FUNCTION_BLOCK TcContinuousAxisCommand IMPLEMENTS itfContinuousAxisCommand
VAR_INPUT
END_VAR
VAR_OUTPUT
END_VAR
VAR
END_VAR

{warning 'add method implementation '}
METHOD Abort : MC_Error
END_METHOD

{warning 'add property implementation'}
PROPERTY Active : BOOL
GET
END_GET
END_PROPERTY

{warning 'add property implementation'}
PROPERTY Busy : BOOL
GET
END_GET
END_PROPERTY

{warning 'add property implementation'}
PROPERTY Command : MC_COMMAND_REF
GET
END_GET
END_PROPERTY

{warning 'add property implementation'}
PROPERTY CommandAborted : BOOL
GET
END_GET
END_PROPERTY

{warning 'add property implementation'}
PROPERTY Done : BOOL
GET
END_GET
END_PROPERTY

{warning 'add property implementation'}
PROPERTY Error : BOOL
GET
END_GET
END_PROPERTY

{warning 'add property implementation'}
PROPERTY ErrorId : MC_Error
GET
END_GET
END_PROPERTY

{warning 'add property implementation'}
PROPERTY InVelocity : BOOL
GET
END_GET
END_PROPERTY

{warning 'add method implementation '}
METHOD Update 		: MC_Error
VAR_INPUT
	Position		: REAL;
	Velocity		: REAL;
	EndVelocity		: REAL;
	Acceleration	: REAL;
	Deceleration	: REAL;
	Jerk			: REAL;
END_VAR
END_METHOD

{warning 'add method implementation '}
METHOD Wait 		: MC_Error (* This method only makes sense in the IEC 61499 environment*)
VAR_INPUT
	Timeout			: TIME;
	AbortOnTimeout	: BOOL;
END_VAR
END_METHOD

END_FUNCTION_BLOCK

(* stored: Version 1.1.0.1, ProductVersion 3.1.4024.12
   POU TcContinuousAxisCommand: Id {2f2c36ee-d9a1-4c99-ab3e-20bd232454f4}, SpecialFunc None
   Method Abort: Id {c3c8fac2-b05c-41e5-8749-a474eccc9071}
   Property Active: Id {e96648dd-1bd3-4a29-b418-6552f02f0ffb}
   Get Get: Id {ac55852b-5e43-4e26-8ddf-130193d08474}
   Property Busy: Id {a79d3a53-e78e-483d-9f5c-125752e7da13}
   Get Get: Id {0e7bd3c9-cfe6-448f-bc0c-793d400ef926}
   Property Command: Id {368f67eb-17a3-499b-b5a0-5540d1977091}
   Get Get: Id {da91f645-ca78-4e17-adce-521510a84717}
   Property CommandAborted: Id {3673eb21-cf48-4174-9543-86f54f9215ff}
   Get Get: Id {80bf0ffa-9357-42e9-a936-54a66f14d60a}
   Property Done: Id {49d4ebe1-1410-45f0-903d-1a70253b1a71}
   Get Get: Id {b618de7e-55c8-48ef-9a70-98d6f499f12f}
   Property Error: Id {f3a5fbb5-5ad3-4f9a-a135-1a57f3fc918a}
   Get Get: Id {6cc312b7-2270-4266-a8ba-66f2bc0be269}
   Property ErrorId: Id {27733607-0b46-4b39-8f5e-84ed640fa1eb}
   Get Get: Id {a71575d9-31f8-4959-8291-2e1de89a864d}
   Property InVelocity: Id {0ff67cb0-fae5-45a9-9909-5f9fb7c4a678}
   Get Get: Id {07ad40ae-31e0-4d8c-b430-5b44d1a9e92f}
   Method Update: Id {3a096b8e-df40-4741-b9d5-725b355372f0}
   Method Wait: Id {36148902-c204-405c-a0dc-9f7051ecc813} *)
